// Mitsubishi GX Works2 project: fbEx02   PLC: Q02/Q02H

PROGRAM MAIN
VAR
  신호점멸_1 : 신호점멸;
END_VAR
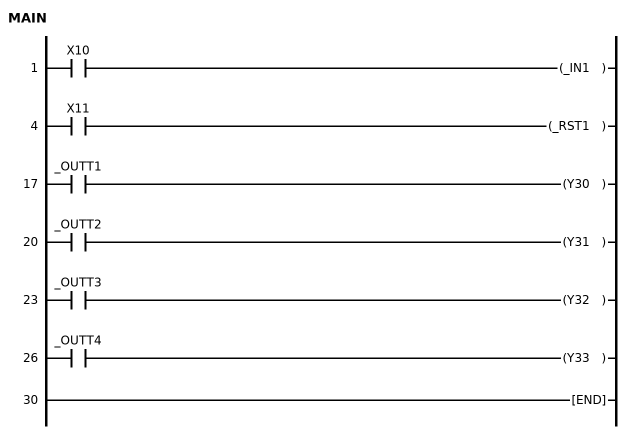
; FB BLK START 신호점멸(신호점멸_1)
1     LD      X10
      OUT     _IN1
4     LD      X11
      OUT     _RST1
; FB START
; FB_NAME 신호점멸
; INSTANCE_NAME 신호점멸_1
; FB IN_B:IN1
; FB OUT_OUTT1:B
; FB IN_B:RST1
; FB OUT_OUTT2:B
; FB OUT_OUTT3:B
; FB OUT_OUTT4:B
; FB END
17    LD      _OUTT1
      OUT     Y30
20    LD      _OUTT2
      OUT     Y31
23    LD      _OUTT3
      OUT     Y32
26    LD      _OUTT4
      OUT     Y33
; FB BLK END
30    END
END_PROGRAM

FUNCTION_BLOCK 신호점멸
VAR_INPUT
  IN1 : BOOL;  (* 입력 *)
  RST1 : BOOL;
END_VAR
VAR
  A_M1 : BOOL;
  T_OUT1 : TIMER;
  T_OUT2 : TIMER;
  T_OUT3 : TIMER;
  T_OUT4 : TIMER;
  A_CNT : COUNTER;
END_VAR
VAR_OUTPUT
  OUTT1 : BOOL;
  OUTT2 : BOOL;
  OUTT3 : BOOL;
  OUTT4 : BOOL;
END_VAR
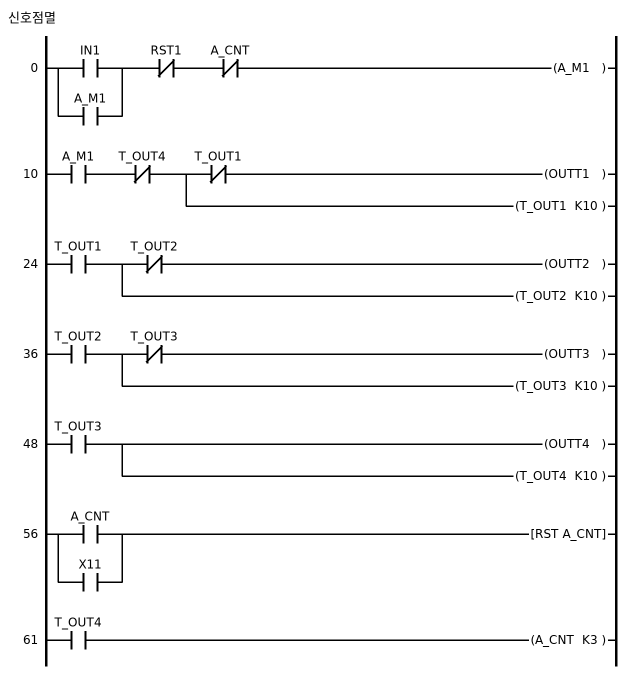
0     LD      IN1
      OR      A_M1
      ANI     RST1
      ANI     A_CNT
      OUT     A_M1
10    LD      A_M1
      ANI     T_OUT4
      MPS
      ANI     T_OUT1
      OUT     OUTT1
      MPP
      OUT     T_OUT1 K10
24    LD      T_OUT1
      MPS
      ANI     T_OUT2
      OUT     OUTT2
      MPP
      OUT     T_OUT2 K10
36    LD      T_OUT2
      MPS
      ANI     T_OUT3
      OUT     OUTT3
      MPP
      OUT     T_OUT3 K10
48    LD      T_OUT3
      OUT     OUTT4
      OUT     T_OUT4 K10
56    LD      A_CNT
      OR      X11
      RST     A_CNT
61    LD      T_OUT4
      OUT     A_CNT K3
END_FUNCTION_BLOCK
